Omron CX-Programmer project NewProject (CX-Programmer 9.70)

# PLC NewPLC1: CP1E E20

## Global symbols (name address type ; comment)
0.01 BOOL  ; stop
100.00 BOOL  ; motor
100.01 BOOL  ; pump

## Program NewProgram1 (cyclic task 0)

### Section Section1

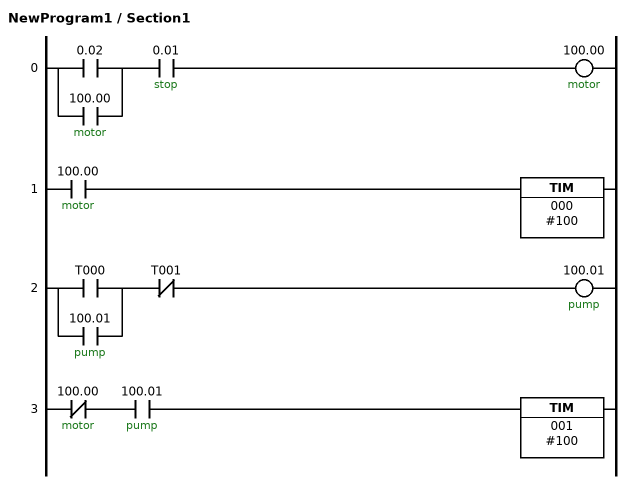
; rung 0
LD 0.02
OR 100.00  ; motor
AND 0.01  ; stop
OUT 100.00  ; motor
; rung 1
LD 100.00  ; motor
TIM 000 #100
; rung 2
LD T000
OR 100.01  ; pump
ANDNOT T001
OUT 100.01  ; pump
; rung 3
LDNOT 100.00  ; motor
AND 100.01  ; pump
TIM 001 #100

### Section END
; rung 0
END(001)